TYPE DUT_AxisCalibration : STRUCT
    reference_position_count      : DINT;
    reference_commutation_angle   : UINT;
    electrical_direction          : INT;
END_STRUCT
END_TYPE

(* stored: Version 1.1.0.1, ProductVersion 3.1.4024.12
   DUT DUT_AxisCalibration: Id {9f95b821-e6f9-4e51-98dd-900047a01006} *)
